// TIA Portal project "BasementLightControl" (V16)
// This program is an implementation of basement light system with 2 switch and 1 light.

(* hardware
DEVICE "S7-1200 station_1"  S7-1200 Station
   slot 0: "Rack_0"  S7-1200 Rack  Rack  V1.0
   slot 1: "PLC_1"  CPU 1211C DC/DC/DC  6ES7 211-1AE40-0XB0  V4.4
DEVICE "TP900 Comfort"  TP900 Comfort
   slot 0: "TP900 Comfort"  TP900 Comfort  6AV2 124-0JC01-0AX0  16.0.0.0
   slot 1: "HMI_RT_5"  TP900 Comfort  6AV2 124-0JC01-0AX0  16.0.0.0
   slot 5: "TP900 Comfort._CP_1"  PROFINET Interface  16.0.0.0
      slot 1: "PROFINET Interface_1"  PROFINET Interface
         slot 1: "Port_1"  Port
         slot 2: "Port_2"  Port
   slot 7: "TP900 Comfort.I/DP_CP_1"  MPI/DP Interface  16.0.0.0
*)

// ===== PLC "PLC_1"  CPU 1211C DC/DC/DC =====

DATA_BLOCK "HMI_Inteface"   // DB1
{ S7_Optimized_Access := 'TRUE' }
VERSION : 0.1
   VAR
      upperSwitch : Bool;   // toggle switch for upper level switch control
      lowerSwitch : Bool;   // toggle switch for lower level switch control
      lightOutput : Bool;   // 0 = Light is ON; 1 = Light is OFF
   END_VAR
BEGIN
END_DATA_BLOCK

DATA_BLOCK "lightControl_DB"   // DB2
{ S7_Optimized_Access := 'TRUE' }
VERSION : 0.1
// stored: InstanceOfName lightControl
"lightControl"
BEGIN
END_DATA_BLOCK

FUNCTION_BLOCK "lightControl"   // FB1, LAD
{ S7_Optimized_Access := 'TRUE' }
VERSION : 0.1
   VAR_INPUT
      UpperLevelSwitch : Bool;
      LowerLevelSwitch : Bool;
   END_VAR
   VAR_OUTPUT
      Light : Bool;
   END_VAR
BEGIN

REGION Network 1: Set Light output when one of the switch is in ON Position
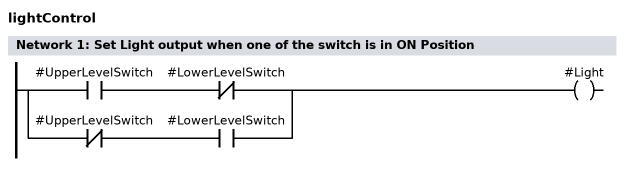
   RUNG wire#powerrail
      Contact( #UpperLevelSwitch )
      I_Contact( #LowerLevelSwitch )
      wire#w1
      Coil( #Light )
   END_RUNG
   RUNG wire#powerrail
      I_Contact( #UpperLevelSwitch )
      Contact( #LowerLevelSwitch )
   END_RUNG wire#w1
   // the same network as SCL:
   #Light := (#UpperLevelSwitch AND NOT #LowerLevelSwitch) OR (NOT #UpperLevelSwitch AND #LowerLevelSwitch);
END_REGION
END_FUNCTION_BLOCK

ORGANIZATION_BLOCK "Main"   // OB1, LAD, ProgramCycle
TITLE = "Main Program Sweep (Cycle)"
{ S7_Optimized_Access := 'TRUE' }
VERSION : 0.1
   VAR_INPUT
      Initial_Call : Bool;   // Initial call of this OB
      Remanence : Bool;   // =True, if remanent data are available
   END_VAR
BEGIN

REGION Network 1: Call Light Control FB
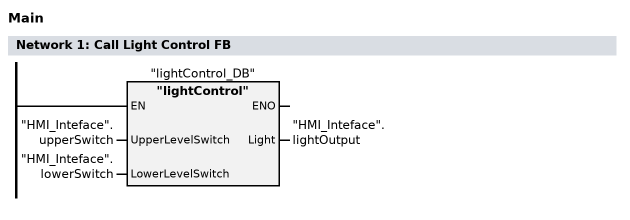
   RUNG wire#powerrail
      "lightControl_DB"(UpperLevelSwitch := "HMI_Inteface".upperSwitch, LowerLevelSwitch := "HMI_Inteface".lowerSwitch, Light => "HMI_Inteface".lightOutput)
   END_RUNG
   // the same network as SCL:
   "lightControl_DB"(UpperLevelSwitch := "HMI_Inteface".upperSwitch,   // "lightControl"
                     LowerLevelSwitch := "HMI_Inteface".lowerSwitch,
                     Light => "HMI_Inteface".lightOutput);
END_REGION
END_ORGANIZATION_BLOCK

(* ===== HMI "HMI_RT_5" =====
system functions are stored by id; their names below are inferred from use
connection "HMI_Connection_7": 
connection "HMI_Connection_1": ETHERNET, S7_1200_OMS

HMI tags "Template"
   "MainNavigationState" : Int, internal
   "SubNavigationState" : Int, internal
   "CurrentUserName" : WString[18], internal
   "DiagState" : Int, internal
   "PopUpBackground" : Bool, internal
   "UserName" : WString[20], internal
   "Password" : WString[20], internal
   "UserIsLoggedIn" : Bool, internal
   "CodeView" : Bool, internal
   "Brightness" : Int, internal
   "CurrentLanguage" : Bool, internal
   "CurrentRecipeName" : WString[30], internal
   "CurrentMachineState" : Int, internal
   "OptionPanelNavigationState" : Int, internal
   "ButtonDown" : Bool, internal
   "ThirdLevelNavigationState" : Int, internal
   "StartScreenName" : WString[60], internal
   "InScreenTabState" : Int, internal
   "DummyTagBool" : Bool, internal
   "DummyTagInt1" : Int, internal
   "DummyTagInt2" : Int, internal
   "DummyTagInt3" : Int, internal
   "DummyDeltaReal" : LReal, internal
   "DummTagReal1" : LReal, internal
   "DummyDeltaInt" : Int, internal

HMI tags "PLC_Tags"
   "HMI_Inteface_upperSwitch" : Bool = PLC HMI_Inteface.upperSwitch, 100 ms
   "HMI_Inteface_lowerSwitch" : Bool = PLC HMI_Inteface.lowerSwitch, 100 ms
   "HMI_Inteface_lightOutput" : Bool = PLC HMI_Inteface.lightOutput, 100 ms

text list "Machine State": 0 'Undefined / Kein Job'; 1 'Production / Produktion'; 2 'Startup / Anlauf'; 3 'Paused / Pausiert'; 4 'Stopped / Gestoppt'; 5 'Shutdown / Beenden'; 6 'Undefined / UNBEKANNT'

text list "timeRange": 1 'Hours / Stunden'; 2 'Days / Tage'; 3 'Weeks / Wochen'; 4 'Months / Monate'; 5 'Years / Jahre'

text list "MachineState_Farfield": 0..1 '???'; 1 'OK'; 2 'ERROR / FEHLER'; 3 'PAUSED / HALT'

text list "Foil Types": 0..1 '120 - 1mm - Transparent'; 1 '120 - 3mm - Transparent'; 2 '240 - 1mm - Transparent'; 3 '240 - 3mm - Transparent'

text list "FunctionState": 0 'Disabled / Deaktiviert'; 1 'Enabled / Aktiviert'

text list "GroundPos": 0 'No / Nein'; 1 'Yes / Ja'

text list "State": 0 'Off / Aus'; 1 'On / An'

graphic list "DiagState": 0 'DiagOkay'; 1 'DiagWarning_1'; 2 'DiagDefault'

graphic list "DiagState_1": 0 'DiagOkay_1'; 1 'DiagWarning'; 2 'DiagDefault'

graphic list "DiagState_2": 0 'DiagOkay_1'; 1 'DiagWarning'; 2 'DiagDefault'

graphic list "DiagState_3": 0 'DiagOkay_White'; 1 'DiagWarning_White'; 2 'Circle'

graphic list "State": 0..1 'OK'; 3 'Error'

graphic list "Machine": 1 'Grafik_Verpackung_Step1_Blink-off'; 2 'Grafik_Verpackung_Step2'; 3 'Grafik_Verpackung_Blink-on'; 6..7 'Grafik_Verpackung_Step1_Blink-off'

screen "20_Messages" 800x480, template "01_One_Nav_Level"
   on GenerateScreen: SetTag("MainNavigationState", 2)
   AlarmView "Alarm view_1" at 0,104 size 800x375
   GraphicView "Graphic view_2" at 0,0 size 800x480; Picture "PopUpBackground"
      Visibility <- "PopUpBackground"

screen "30_Diagnostics" 800x480, template "01_One_Nav_Level"
   on GenerateScreen: SetTag("MainNavigationState", 3)
   SysDiagControl "System diagnostics view_1" at 0,104 size 800x375
   GraphicView "Graphic view_2" at 0,0 size 800x480; Picture "PopUpBackground"
      Visibility <- "PopUpBackground"

screen "40_Settings" 800x480, template "02_Settings"
   on GenerateScreen: SetTag("MainNavigationState", 4)
   Slider "Template_Slider_1" at 320,133 size 300x30; Caption 'SIMATIC'
      on Change: function_e4c2bb66("Brightness")
      ProcessValue <- "Brightness"
   TextField "Template_Text field_1" at 180,136 size 92x24; Text 'Brightness / Helligkeit'
   GraphicView "Graphic view_2" at 0,0 size 800x480; Picture "PopUpBackground"
      Visibility <- "PopUpBackground"

screen "10_Startscreen" 800x480, template "01_One_Nav_Level"
   on GenerateScreen: "GetStartScreenName"(); "CheckCurrentUserName"(); SetTag("MainNavigationState", 1)
   GraphicView "Graphic view_2" at 0,0 size 800x480; Picture "PopUpBackground"
      Visibility <- "PopUpBackground"
   GraphicView "Graphic view_4" at 276,110 size 76x90; Picture "lighton"
      Visibility <- "HMI_Inteface_lightOutput"
   GraphicView "Graphic view_1" at 115,128 size 566x347; Picture "Stairs"
   Switch "Switch_1" at 10,108 size 64x169; CaptionText 'Upper'; TextOff 'OFF'; TextOn 'ON'
      ProcessValue <- "HMI_Inteface_upperSwitch"
   Switch "Switch_2" at 730,306 size 64x169; TextOn 'ON'; CaptionText 'Bottom'; TextOff 'OFF'
      ProcessValue <- "HMI_Inteface_lowerSwitch"
   GraphicView "Graphic view_3" at 276,110 size 76x90; Picture "lightoff"
      Visibility <- "HMI_Inteface_lightOutput"
   GraphicView "Graphic view_5" at 409,110 size 76x90; Picture "lighton"
      Visibility <- "HMI_Inteface_lightOutput"
   GraphicView "Graphic view_6" at 542,110 size 76x90; Picture "lighton"
      Visibility <- "HMI_Inteface_lightOutput"
   GraphicView "Graphic view_7" at 409,110 size 76x90; Picture "lightoff"
      Visibility <- "HMI_Inteface_lightOutput"
   GraphicView "Graphic view_8" at 542,110 size 76x90; Picture "lightoff"
      Visibility <- "HMI_Inteface_lightOutput"

Template "02_Two_Nav_Levels" 800x480
   GraphicView "gfxPrevScreenIcon" at 760,444 size 24x24; Picture "PrevScreen_Icon"
   Button "btnSubNav1" at 0,432 size 120x48; TextOff 'Overview / Übersicht'
      on Click: SetTag("SubNavigationState", 1)
   Button "btnSubNav2" at 120,432 size 120x48; TextOff 'Module 1 / Modul 1'
      on Click: SetTag("SubNavigationState", 2)
   Button "btnSubNav3" at 240,432 size 120x48; TextOff 'Module 2 / Modul 2'
      on Click: SetTag("SubNavigationState", 3)
   Button "btnSubNav4" at 360,432 size 120x48; TextOff 'Module 3 / Modul 3'
      on Click: SetTag("SubNavigationState", 4)
   Button "btnSubNav5" at 480,432 size 120x48; TextOff 'Module 4 / Modul 4'
      on Click: SetTag("SubNavigationState", 5)
   Button "btnSubNav6" at 600,432 size 120x48; TextOff 'Module 5 / Modul 5'
      on Click: SetTag("SubNavigationState", 6)
   Button "btnPreviousScreen" at 744,432 size 56x48; TextOff 'Text'
      on Click: function_efd93a16()
   Gauge "gaugeDiagStateUpdate" at 566,2 size 50x50; CaptionText 'SIMATIC'
      on Change: "CheckDiagState"()
      ProcessValue <- "@DiagnosticsIndicatorTag"
   TextField "txtTitleBar" at 16,8 size 495x32; Text 'Basement Light Control / Applikation'
   GraphicView "gfxNavigationIcon" at 761,15 size 23x19; Picture "Hamburger_Icon"
   Button "btnNavigation" at 744,0 size 56x48; TextOff 'Text'
      on Click: function_cf6f4242("GraphX_Slidein_Right", 1)
   TextField "txtStateHeadline" at 75,55 size 123x23; Text 'State / Status'
   TextField "txtRecipeHeadline" at 281,55 size 154x23; Text 'Current Recipe / Rezeptur'
   TextField "txtOperatorHeadline" at 527,55 size 129x23; Text 'Operator / Bediener'
   SymbolicIOField "ioState" at 75,72 size 119x30; TextOn '1'; TextOff '0'; TextList "Machine State"
      ProcessValue <- "CurrentMachineState"
   IOField "ioRecipe" at 281,72 size 158x30; FormatPattern ??????????????????????????????
      ProcessValue <- "CurrentRecipeName"
   IOField "ioOperator" at 527,72 size 126x30; FormatPattern ??????????????????
      ProcessValue <- "CurrentUserName"
   Button "btnState" at 202,56 size 40x40; TextOff '...'; PictureOff "More_Icon"
      on Click: "ShowOperatingModePopUp"()
   Button "btnRecipe" at 449,56 size 40x40; TextOff '...'; PictureOff "More_Icon"
      on Click: "ShowRecipePopUp"()
   Rectangle "rectState" at 0,48 size 56x56
      Appearance <- "CurrentMachineState"
   Rectangle "rectSystemDiagnosticsIndicator" at 744,48 size 56x56
      Appearance <- "DiagState"
   GraphicIOField "gioDiagState" at 756,60 size 32x32; PictureList "DiagState_3"
      ProcessValue <- "DiagState"
   Button "btnDiagState" at 744,48 size 56x56; TextOff 'Text'
      on Click: ActivateScreen("30_Diagnostics", 0)
   Button "btnOperator" at 669,56 size 40x40; TextOff '...'; PictureOff "More_Icon"
      on Click: "ShowLoginPopUp"()
   Button "btnStartscreen" at 0,0 size 250x45; TextOff 'Text'
      on Click: "ActivateStartScreen"()
   Button "btnSubNavActive1" at 0,432 size 120x48; TextOff 'Overview / Übersicht'
      Visibility <- "SubNavigationState"
   Button "btnSubNavActive2" at 120,432 size 120x48; TextOff 'Module 1 / Modul 1'
      Visibility <- "SubNavigationState"
   Button "btnSubNavActive3" at 240,432 size 120x48; TextOff 'Module 2 / Modul 2'
      Visibility <- "SubNavigationState"
   Button "btnSubNavActive4" at 360,432 size 120x48; TextOff 'Module 3 / Modul 3'
      Visibility <- "SubNavigationState"
   Button "btnSubNavActive5" at 480,432 size 120x48; TextOff 'Module 4 / Modul 4'
      Visibility <- "SubNavigationState"
   Button "btnSubNavActive6" at 600,432 size 120x48; TextOff 'Module 5 / Modul 5'
      Visibility <- "SubNavigationState"
   Rectangle "rectIndicatorActive1" at 0,475 size 120x5
      Visibility <- "SubNavigationState"
   Rectangle "rectIndicatorActive2" at 120,475 size 120x5
      Visibility <- "SubNavigationState"
   Rectangle "rectIndicatorActive3" at 240,475 size 120x5
      Visibility <- "SubNavigationState"
   Rectangle "rectIndicatorActive4" at 360,475 size 120x5
      Visibility <- "SubNavigationState"
   Rectangle "rectIndicatorActive5" at 480,475 size 120x5
      Visibility <- "SubNavigationState"
   Rectangle "rectIndicatorActive6" at 600,475 size 120x5
      Visibility <- "SubNavigationState"

Template "03_Three_Nav_Levels" 800x480
   Button "btnStartscreen" at 0,0 size 326x45; TextOff 'Text'
      on Click: "ActivateStartScreen"()
   Gauge "gaugeDiagStateUpdate" at 566,2 size 50x50; CaptionText 'SIMATIC'
      on Change: "CheckDiagState"()
      ProcessValue <- "@DiagnosticsIndicatorTag"
   TextField "txtTitleBar" at 16,8 size 495x32; Text 'Basement Light Control / Applikation'
   GraphicView "gfxNavigationIcon" at 761,15 size 23x19; Picture "Hamburger_Icon"
   Button "btnNavigation" at 744,0 size 56x48; TextOff 'Text'
      on Click: function_cf6f4242("GraphX_Slidein_Right", 1)
   Rectangle "rectSystemDiagnosticsIndicator" at 744,48 size 56x56
      Appearance <- "DiagState"
   GraphicIOField "gioDiagState" at 756,60 size 32x32; PictureList "DiagState_3"
      ProcessValue <- "DiagState"
   Button "btnDiagState" at 744,48 size 56x56; TextOff 'Text'
      on Click: ActivateScreen("30_Diagnostics", 0)
   TextField "txtStateHeadline" at 75,55 size 123x23; Text 'State / Status'
   TextField "txtOperatorHeadline" at 527,55 size 129x23; Text 'Operator / Bediener'
   SymbolicIOField "ioState" at 75,72 size 119x30; TextOn '1'; TextOff '0'; TextList "Machine State"
      ProcessValue <- "CurrentMachineState"
   IOField "ioOperator" at 527,72 size 126x30; FormatPattern ??????????????????
      ProcessValue <- "CurrentUserName"
   Button "btnState" at 202,56 size 40x40; TextOff '...'; PictureOff "More_Icon"
      on Click: "ShowOperatingModePopUp"()
   Button "btnOperator" at 669,56 size 40x40; TextOff '...'; PictureOff "More_Icon"
      on Click: "ShowLoginPopUp"()
   Rectangle "rectState" at 0,48 size 56x56
      Appearance <- "CurrentMachineState"
   TextField "txtRecipeHeadline" at 281,55 size 154x23; Text 'Current Recipe / Rezeptur'
   IOField "ioRecipe" at 281,72 size 158x30; FormatPattern ??????????????????????????????
      ProcessValue <- "CurrentRecipeName"
   Button "btnRecipe" at 449,56 size 40x40; TextOff '...'; PictureOff "More_Icon"
      on Click: "ShowRecipePopUp"()
   Button "btnThirdLevel4btnOff1" at 0,104 size 56x83; TextOff 'Text'
   Button "btnThirdLevel4btnOff2" at 0,186 size 56x83; TextOff 'Text'
   Button "btnThirdLevel4btnOff3" at 0,268 size 56x83; TextOff 'Text'
   Button "btnThirdLevel4btnOff4" at 0,350 size 56x82; TextOff 'Text'
   Button "btnThirdLevel4btnOn1" at 0,187 size 56x81; TextOff 'Text'
      Visibility <- "ThirdLevelNavigationState"
   Button "btnThirdLevel4btnOn2" at 0,104 size 56x82; TextOff 'Text'
      Visibility <- "ThirdLevelNavigationState"
   Button "btnThirdLevel4btnOn3" at 0,269 size 56x81; TextOff 'Text'
      Visibility <- "ThirdLevelNavigationState"
   Button "btnThirdLevel4btnOn4" at 0,351 size 56x81; TextOff 'Text'
      Visibility <- "ThirdLevelNavigationState"
   Rectangle "rectIndicator4btnActive1" at 0,104 size 5x82
      Visibility <- "ThirdLevelNavigationState"
   Rectangle "rectIndicator4btnActive2" at 0,187 size 5x81
      Visibility <- "ThirdLevelNavigationState"
   Rectangle "rectIndicator4btnActive3" at 0,269 size 5x81
      Visibility <- "ThirdLevelNavigationState"
   Rectangle "rectIndicator4btnActive4" at 0,351 size 5x81
      Visibility <- "ThirdLevelNavigationState"
   Button "btnSubNav1" at 0,432 size 120x48; TextOff 'Overview / Übersicht'
      on Click: SetTag("SubNavigationState", 1)
   Button "btnSubNav2" at 120,432 size 120x48; TextOff 'Module 1 / Modul 1'
      on Click: SetTag("SubNavigationState", 2)
   Button "btnSubNav3" at 240,432 size 120x48; TextOff 'Module 2 / Modul 2'
      on Click: SetTag("SubNavigationState", 3)
   Button "btnSubNav4" at 360,432 size 120x48; TextOff 'Module 3 / Modul 3'
      on Click: SetTag("SubNavigationState", 4)
   Button "btnSubNav5" at 480,432 size 120x48; TextOff 'Module 4 / Modul 4'
      on Click: SetTag("SubNavigationState", 5)
   Button "btnSubNav6" at 600,432 size 120x48; TextOff 'Module 5 / Modul 5'
      on Click: SetTag("SubNavigationState", 6)
   GraphicView "gfxPrevScreenIcon" at 760,444 size 24x24; Picture "PrevScreen_Icon"
   Button "btnPreviousScreen" at 744,432 size 56x48; TextOff 'Text'
      on Click: function_efd93a16()
   Button "btnSubNavActive1" at 0,432 size 120x48; TextOff 'Overview / Übersicht'
      Visibility <- "SubNavigationState"
   Button "btnSubNavActive2" at 120,432 size 120x48; TextOff 'Module 1 / Modul 1'
      Visibility <- "SubNavigationState"
   Button "btnSubNavActive3" at 240,432 size 120x48; TextOff 'Module 2 / Modul 2'
      Visibility <- "SubNavigationState"
   Button "btnSubNavActive4" at 360,432 size 120x48; TextOff 'Module 3 / Modul 3'
      Visibility <- "SubNavigationState"
   Button "btnSubNavActive5" at 480,432 size 120x48; TextOff 'Module 4 / Modul 4'
      Visibility <- "SubNavigationState"
   Button "btnSubNavActive6" at 600,432 size 120x48; TextOff 'Module 5 / Modul 5'
      Visibility <- "SubNavigationState"
   Rectangle "rectIndicatorActive1" at 0,475 size 120x5
      Visibility <- "SubNavigationState"
   Rectangle "rectIndicatorActive2" at 120,475 size 120x5
      Visibility <- "SubNavigationState"
   Rectangle "rectIndicatorActive3" at 240,475 size 120x5
      Visibility <- "SubNavigationState"
   Rectangle "rectIndicatorActive4" at 360,475 size 120x5
      Visibility <- "SubNavigationState"
   Rectangle "rectIndicatorActive5" at 480,475 size 120x5
      Visibility <- "SubNavigationState"
   Rectangle "rectIndicatorActive6" at 600,475 size 120x5
      Visibility <- "SubNavigationState"

Template "03_Three_Nav_Levels_w_OptionPanel" 800x480
   Button "btnStartscreen" at 0,0 size 326x45; TextOff 'Text'
      on Click: "ActivateStartScreen"()
   Gauge "gaugeDiagStateUpdate" at 566,2 size 50x50; CaptionText 'SIMATIC'
      on Change: "CheckDiagState"()
      ProcessValue <- "@DiagnosticsIndicatorTag"
   TextField "txtTitleBar" at 16,8 size 495x32; Text 'Basement Light Control / Applikation'
   GraphicView "gfxNavigationIcon" at 761,15 size 23x19; Picture "Hamburger_Icon"
   Button "btnNavigation" at 744,0 size 56x48; TextOff 'Text'
      on Click: function_cf6f4242("GraphX_Slidein_Right", 1)
   Rectangle "rectSystemDiagnosticsIndicator" at 744,48 size 56x56
      Appearance <- "DiagState"
   GraphicIOField "gioDiagState" at 756,60 size 32x32; PictureList "DiagState_3"
      ProcessValue <- "DiagState"
   Button "btnDiagState" at 744,48 size 56x56; TextOff 'Text'
      on Click: ActivateScreen("30_Diagnostics", 0)
   TextField "txtStateHeadline" at 75,55 size 123x23; Text 'State / Status'
   TextField "txtOperatorHeadline" at 527,55 size 129x23; Text 'Operator / Bediener'
   SymbolicIOField "ioState" at 75,72 size 119x30; TextOn '1'; TextOff '0'; TextList "Machine State"
      ProcessValue <- "CurrentMachineState"
   IOField "ioOperator" at 527,72 size 126x30; FormatPattern ??????????????????
      ProcessValue <- "CurrentUserName"
   Button "btnState" at 202,56 size 40x40; TextOff '...'; PictureOff "More_Icon"
      on Click: "ShowOperatingModePopUp"()
   Button "btnOperator" at 669,56 size 40x40; TextOff '...'; PictureOff "More_Icon"
      on Click: "ShowLoginPopUp"()
   Rectangle "rectState" at 0,48 size 56x56
      Appearance <- "CurrentMachineState"
   TextField "txtRecipeHeadline" at 281,55 size 154x23; Text 'Current Recipe / Rezeptur'
   IOField "ioRecipe" at 281,72 size 158x30; FormatPattern ??????????????????????????????
      ProcessValue <- "CurrentRecipeName"
   Button "btnRecipe" at 449,56 size 40x40; TextOff '...'; PictureOff "More_Icon"
      on Click: "ShowRecipePopUp"()
   Button "btnThirdLevelOff1" at 0,104 size 56x83; TextOff 'Text'
   Button "btnThirdLevelOff2" at 0,186 size 56x83; TextOff 'Text'
   Button "btnThirdLevelOff3" at 0,268 size 56x83; TextOff 'Text'
   Button "btnThirdLevelOff4" at 0,350 size 56x82; TextOff 'Text'
   Button "btnThirdLevelOn1" at 0,187 size 56x81; TextOff 'Text'
      Visibility <- "ThirdLevelNavigationState"
   Button "btnThirdLevelOn2" at 0,104 size 56x82; TextOff 'Text'
      Visibility <- "ThirdLevelNavigationState"
   Button "btnThirdLevelOn3" at 0,269 size 56x81; TextOff 'Text'
      Visibility <- "ThirdLevelNavigationState"
   Button "btnThirdLevelOn4" at 0,351 size 56x81; TextOff 'Text'
      Visibility <- "ThirdLevelNavigationState"
   Rectangle "rectIndicatorActive1_1" at 0,104 size 5x82
      Visibility <- "ThirdLevelNavigationState"
   Rectangle "rectIndicatorActive1_2" at 0,187 size 5x81
      Visibility <- "ThirdLevelNavigationState"
   Rectangle "rectIndicatorActive1_3" at 0,269 size 5x81
      Visibility <- "ThirdLevelNavigationState"
   Rectangle "rectIndicatorActive1_4" at 0,351 size 5x81
      Visibility <- "ThirdLevelNavigationState"
   Button "btnOption1btn1" at 744,104 size 56x328; TextOff 'Text'; PictureOff "ManFunctions_Off"; PictureOn "ManFunctions_Off"
      on Click: "ShowOptionPanelPopUp"()
   Button "btnSubNav1" at 0,432 size 120x48; TextOff 'Overview / Übersicht'
      on Click: SetTag("SubNavigationState", 1)
   Button "btnSubNav2" at 120,432 size 120x48; TextOff 'Module 1 / Modul 1'
      on Click: SetTag("SubNavigationState", 2)
   Button "btnSubNav3" at 240,432 size 120x48; TextOff 'Module 2 / Modul 2'
      on Click: SetTag("SubNavigationState", 3)
   Button "btnSubNav4" at 360,432 size 120x48; TextOff 'Module 3 / Modul 3'
      on Click: SetTag("SubNavigationState", 4)
   Button "btnSubNav5" at 480,432 size 120x48; TextOff 'Module 4 / Modul 4'
      on Click: SetTag("SubNavigationState", 5)
   Button "btnSubNav6" at 600,432 size 120x48; TextOff 'Module 5 / Modul 5'
      on Click: SetTag("SubNavigationState", 6)
   GraphicView "gfxPrevScreenIcon" at 760,444 size 24x24; Picture "PrevScreen_Icon"
   Button "btnPreviousScreen" at 744,432 size 56x48; TextOff 'Text'
      on Click: function_efd93a16()
   Button "btnSubNavActive1" at 0,432 size 120x48; TextOff 'Overview / Übersicht'
      Visibility <- "SubNavigationState"
   Button "btnSubNavActive2" at 120,432 size 120x48; TextOff 'Module 1 / Modul 1'
      Visibility <- "SubNavigationState"
   Button "btnSubNavActive3" at 240,432 size 120x48; TextOff 'Module 2 / Modul 2'
      Visibility <- "SubNavigationState"
   Button "btnSubNavActive4" at 360,432 size 120x48; TextOff 'Module 3 / Modul 3'
      Visibility <- "SubNavigationState"
   Button "btnSubNavActive5" at 480,432 size 120x48; TextOff 'Module 4 / Modul 4'
      Visibility <- "SubNavigationState"
   Button "btnSubNavActive6" at 600,432 size 120x48; TextOff 'Module 5 / Modul 5'
      Visibility <- "SubNavigationState"
   Rectangle "rectIndicatorActive1" at 0,475 size 120x5
      Visibility <- "SubNavigationState"
   Rectangle "rectIndicatorActive2" at 120,475 size 120x5
      Visibility <- "SubNavigationState"
   Rectangle "rectIndicatorActive3" at 240,475 size 120x5
      Visibility <- "SubNavigationState"
   Rectangle "rectIndicatorActive4" at 360,475 size 120x5
      Visibility <- "SubNavigationState"
   Rectangle "rectIndicatorActive5" at 480,475 size 120x5
      Visibility <- "SubNavigationState"
   Rectangle "rectIndicatorActive6" at 600,475 size 120x5
      Visibility <- "SubNavigationState"

Template "01_One_Nav_Level" 800x480
   Rectangle "rectSystemDiagnosticsIndicator" at 744,48 size 56x56
      Appearance <- "DiagState"
   GraphicIOField "gioDiagState" at 756,60 size 32x32; PictureList "DiagState_3"
      ProcessValue <- "DiagState"
   Button "btnDiagState" at 744,48 size 56x56; TextOff 'Text'
      on Click: ActivateScreen("30_Diagnostics", 0)
   TextField "txtStateHeadline" at 75,55 size 123x23; Text 'State / Status'
   TextField "txtOperatorHeadline" at 527,55 size 129x23; Text 'Operator / Bediener'
   SymbolicIOField "ioState" at 75,72 size 119x30; TextOn '1'; TextOff '0'; TextList "Machine State"
      ProcessValue <- "CurrentMachineState"
   IOField "ioOperator" at 527,72 size 126x30; FormatPattern ??????????????????
      ProcessValue <- "CurrentUserName"
   Button "btnState" at 202,56 size 40x40; TextOff '...'; PictureOff "More_Icon"
      on Click: "ShowOperatingModePopUp"()
   Button "btnOperator" at 669,56 size 40x40; TextOff '...'; PictureOff "More_Icon"
      on Click: "ShowLoginPopUp"()
   Rectangle "rectState" at 0,48 size 56x56
      Appearance <- "CurrentMachineState"
   TextField "txtRecipeHeadline" at 281,55 size 154x23; Text 'Current Recipe / Rezeptur'
   IOField "ioRecipe" at 281,72 size 158x30; FormatPattern ??????????????????????????????
      ProcessValue <- "CurrentRecipeName"
   Button "btnRecipe" at 449,56 size 40x40; TextOff '...'; PictureOff "More_Icon"
      on Click: "ShowRecipePopUp"()
   Gauge "gaugeDiagStateUpdate" at 566,2 size 50x50; CaptionText 'SIMATIC'
      on Change: "CheckDiagState"()
      ProcessValue <- "@DiagnosticsIndicatorTag"
   GraphicView "gfxNavigationIcon" at 761,15 size 23x19; Picture "Hamburger_Icon"
   Button "btnNavigation" at 744,0 size 56x48; TextOff 'Text'
      on Click: function_cf6f4242("GraphX_Slidein_Right", 1)
   TextField "txtTitleBar" at 16,8 size 495x32; Text 'Basement Light Control / Applikation'
   Button "btnStartscreen" at 0,0 size 250x45; TextOff 'Text'
      on Click: "ActivateStartScreen"()

Template "02_Two_Nav_Levels_Large_Text" 800x480
   Gauge "gaugeDiagStateUpdate" at 566,2 size 50x50; CaptionText 'SIMATIC'
      on Change: "CheckDiagState"()
      ProcessValue <- "@DiagnosticsIndicatorTag"
   TextField "txtTitleBar" at 16,8 size 495x32; Text 'Basement Light Control / Applikation'
   GraphicView "gfxNavigationIcon" at 761,15 size 23x19; Picture "Hamburger_Icon"
   Button "btnNavigation" at 744,0 size 56x48; TextOff 'Text'
      on Click: function_cf6f4242("GraphX_Slidein_Right", 1)
   TextField "txtStateHeadline" at 75,55 size 123x23; Text 'State / Status'
   TextField "txtRecipeHeadline" at 281,55 size 154x23; Text 'Current Recipe / Rezeptur'
   TextField "txtOperatorHeadline" at 527,55 size 129x23; Text 'Operator / Bediener'
   SymbolicIOField "ioState" at 75,72 size 119x30; TextOn '1'; TextOff '0'; TextList "Machine State"
      ProcessValue <- "CurrentMachineState"
   IOField "ioRecipe" at 281,72 size 158x30; FormatPattern ??????????????????????????????
      ProcessValue <- "CurrentRecipeName"
   IOField "ioOperator" at 527,72 size 126x30; FormatPattern ??????????????????
      ProcessValue <- "CurrentUserName"
   Button "btnState" at 202,56 size 40x40; TextOff '...'; PictureOff "More_Icon"
      on Click: "ShowOperatingModePopUp"()
   Button "btnRecipe" at 449,56 size 40x40; TextOff '...'; PictureOff "More_Icon"
      on Click: "ShowRecipePopUp"()
   Rectangle "rectState" at 0,48 size 56x56
      Appearance <- "CurrentMachineState"
   GraphicView "gfxPrevScreenIcon" at 760,444 size 24x24; Picture "PrevScreen_Icon"
   Button "btnPreviousScreen" at 744,432 size 56x48; TextOff 'Text'
      on Click: function_efd93a16()
   TextField "txtCurrentStateInfo" at 16,444 size 505x24; Text 'Optional Text about current state / Optional. Text aktueller Status'
   Rectangle "rectSystemDiagnosticsIndicator" at 744,48 size 56x56
      Appearance <- "DiagState"
   GraphicIOField "gioDiagState" at 756,60 size 32x32; PictureList "DiagState_3"
      ProcessValue <- "DiagState"
   Button "btnDiagState" at 744,48 size 56x56; TextOff 'Text'
      on Click: ActivateScreen("30_Diagnostics", 0)
   Button "btnOperator" at 669,56 size 40x40; TextOff '...'; PictureOff "More_Icon"
      on Click: "ShowLoginPopUp"()
   Button "btnStartscreen" at 0,0 size 250x45; TextOff 'Text'
      on Click: "ActivateStartScreen"()
   Rectangle "rectSubNavigation1" at 0,104 size 264x83
      Appearance <- "ThirdLevelNavigationState"
   Rectangle "rectSubNavigation2" at 0,186 size 264x83
      Appearance <- "ThirdLevelNavigationState"
   Rectangle "rectSubNavigation3" at 0,268 size 264x83
      Appearance <- "ThirdLevelNavigationState"
   Rectangle "rectSubNavigation4" at 0,350 size 264x82
      Appearance <- "ThirdLevelNavigationState"
   TextField "txtOption1" at 16,120 size 232x24; Text 'Option 1'
   IOField "ioValueOption1" at 16,152 size 236x24; FormatPattern ??????????????????????????????????????????????????
   TextField "txtOption2" at 16,202 size 232x24; Text 'Option 2'
   IOField "ioValueOption2" at 16,234 size 236x24; FormatPattern ??????????????????????????????????????????????????
   TextField "txtOption3" at 16,284 size 232x24; Text 'Option 3'
   IOField "ioValueOption3" at 16,316 size 236x24; FormatPattern ??????????????????????????????????????????????????
   TextField "txtOption4" at 16,366 size 232x24; Text 'Option 4'
   IOField "ioValueOption4" at 16,398 size 236x24; FormatPattern ??????????????????????????????????????????????????
   Button "btnSubNavigation1" at 0,104 size 264x83; TextOff 'Text'
      on Click: SetTag("ThirdLevelNavigationState", 1)
   Button "btnSubNavigation2" at 0,186 size 264x83; TextOff 'Text'
      on Click: SetTag("ThirdLevelNavigationState", 2)
   Button "btnSubNavigation3" at 0,268 size 264x83; TextOff 'Text'
      on Click: SetTag("ThirdLevelNavigationState", 3)
   Button "btnSubNavigation4" at 0,350 size 264x83; TextOff 'Text'
      on Click: SetTag("ThirdLevelNavigationState", 4)

Template "02_Two_Nav_Levels_Text" 800x480
   Button "btnSubNav1" at 0,120 size 136x56; TextOn 'Item 1'; TextOff 'Item 1'
      on Click: SetTag("SubNavigationState", 1)
   Button "btnSubNav2" at 0,175 size 136x56; TextOn 'Item 2'; TextOff 'Item 2'
      on Click: SetTag("SubNavigationState", 2)
   Button "btnSubNav3" at 0,230 size 136x60; TextOn 'Item 3'; TextOff 'Item 3'
      on Click: SetTag("SubNavigationState", 3)
   GraphicView "gfxRuntimeStop" at 57,443 size 23x28; Picture "Power_dark"
   Button "btnRuntimeStop" at 0,432 size 136x48; TextOff 'Text'
      on Click: StopRuntime(0)
   Button "btnSubNav3_1" at 0,289 size 136x60; TextOn 'Item 4'; TextOff 'Item 4'
      on Click: SetTag("SubNavigationState", 4)
   Button "btnSubNav3_2" at 0,348 size 136x60; TextOn 'Item 5'; TextOff 'Item 5'
      on Click: SetTag("SubNavigationState", 5)
   Button "btnSubNavActive3" at 0,230 size 136x60; TextOff 'Item 3'
      Visibility <- "SubNavigationState"
   Button "btnSubNavActive1" at 0,120 size 136x56; TextOff 'Item 1'
      Visibility <- "SubNavigationState"
   Button "btnSubNavActive2" at 0,175 size 136x56; TextOff 'Item 2'
      Visibility <- "SubNavigationState"
   Rectangle "rectIndicatorActive3" at 0,230 size 5x60
      Visibility <- "SubNavigationState"
   Rectangle "rectIndicatorActive1" at 0,120 size 5x56
      Visibility <- "SubNavigationState"
   Rectangle "rectIndicatorActive2" at 0,175 size 5x56
      Visibility <- "SubNavigationState"
   Button "btnSubNavActive3_1" at 0,290 size 136x60; TextOff 'Item 4'
      Visibility <- "SubNavigationState"
   Rectangle "rectIndicatorActive3_1" at 0,290 size 5x60
      Visibility <- "SubNavigationState"
   Button "btnSubNavActive3_2" at 0,350 size 136x60; TextOff 'Item 5'
      Visibility <- "SubNavigationState"
   Rectangle "rectIndicatorActive3_2" at 0,350 size 5x60
      Visibility <- "SubNavigationState"
   Gauge "gaugeDiagStateUpdate" at 566,2 size 50x50; CaptionText 'SIMATIC'
      on Change: "CheckDiagState"()
      ProcessValue <- "@DiagnosticsIndicatorTag"
   GraphicView "gfxNavigationIcon" at 761,15 size 23x19; Picture "Hamburger_Icon"
   Button "btnNavigation" at 744,0 size 56x48; TextOff 'Text'
      on Click: function_cf6f4242("GraphX_Slidein_Right", 1)
   TextField "txtTitleBar" at 16,8 size 495x32; Text 'Basement Light Control / Applikation'
   Button "btnStartscreen" at 0,0 size 250x45; TextOff 'Text'
      on Click: "ActivateStartScreen"()
   TextField "txtStateHeadline" at 75,55 size 123x23; Text 'State / Status'
   TextField "txtOperatorHeadline" at 527,55 size 129x23; Text 'Operator / Bediener'
   SymbolicIOField "ioState" at 75,72 size 119x30; TextOn '1'; TextOff '0'; TextList "Machine State"
      ProcessValue <- "CurrentMachineState"
   IOField "ioOperator" at 527,72 size 126x30; FormatPattern ??????????????????
      ProcessValue <- "CurrentUserName"
   Button "btnState" at 202,56 size 40x40; TextOff '...'; PictureOff "More_Icon"
      on Click: "ShowOperatingModePopUp"()
   Button "btnOperator" at 669,56 size 40x40; TextOff '...'; PictureOff "More_Icon"
      on Click: "ShowLoginPopUp"()
   Rectangle "rectState" at 0,48 size 56x56
      Appearance <- "CurrentMachineState"
   TextField "txtRecipeHeadline" at 281,55 size 154x23; Text 'Current Recipe / Rezeptur'
   IOField "ioRecipe" at 281,72 size 158x30; FormatPattern ??????????????????????????????
      ProcessValue <- "CurrentRecipeName"
   Button "btnRecipe" at 449,56 size 40x40; TextOff '...'; PictureOff "More_Icon"
      on Click: "ShowRecipePopUp"()
   Rectangle "rectSystemDiagnosticsIndicator" at 744,48 size 56x56
      Appearance <- "DiagState"
   GraphicIOField "gioDiagState" at 756,60 size 32x32; PictureList "DiagState_3"
      ProcessValue <- "DiagState"
   Button "btnDiagState" at 744,48 size 56x56; TextOff 'Text'
      on Click: ActivateScreen("30_Diagnostics", 0)

Template "02_Settings" 800x480
   Button "btnSubNav1" at 0,120 size 136x56; TextOn 'Display'; TextOff 'Display'
      on Click: SetTag("SubNavigationState", 1)
   GraphicView "gfxRuntimeStop" at 57,443 size 23x28; Picture "Power_dark"
   Button "btnRuntimeStop" at 0,432 size 136x48; TextOff 'Text'
      on Click: StopRuntime(0)
   Button "btnSubNavActive1" at 0,120 size 136x56; TextOn 'Display'; TextOff 'Display'
      Visibility <- "SubNavigationState"
   Rectangle "rectIndicatorActive1" at 0,120 size 5x56
      Visibility <- "SubNavigationState"
   Gauge "gaugeDiagStateUpdate" at 566,2 size 50x50; CaptionText 'SIMATIC'
      on Change: "CheckDiagState"()
      ProcessValue <- "@DiagnosticsIndicatorTag"
   GraphicView "gfxNavigationIcon" at 761,15 size 23x19; Picture "Hamburger_Icon"
   Button "btnNavigation" at 744,0 size 56x48; TextOff 'Text'
      on Click: function_cf6f4242("GraphX_Slidein_Right", 1)
   TextField "txtTitleBar" at 16,8 size 495x32; Text 'Basement Light Control / Applikation'
   Button "btnStartscreen" at 0,0 size 250x45; TextOff 'Text'
      on Click: "ActivateStartScreen"()
   TextField "txtStateHeadline" at 75,55 size 123x23; Text 'State / Status'
   TextField "txtOperatorHeadline" at 527,55 size 129x23; Text 'Operator / Bediener'
   SymbolicIOField "ioState" at 75,72 size 119x30; TextOn '1'; TextOff '0'; TextList "Machine State"
      ProcessValue <- "CurrentMachineState"
   IOField "ioOperator" at 527,72 size 126x30; FormatPattern ??????????????????
      ProcessValue <- "CurrentUserName"
   Button "btnState" at 202,56 size 40x40; TextOff '...'; PictureOff "More_Icon"
      on Click: "ShowOperatingModePopUp"()
   Button "btnOperator" at 669,56 size 40x40; TextOff '...'; PictureOff "More_Icon"
      on Click: "ShowLoginPopUp"()
   Rectangle "rectState" at 0,48 size 56x56
      Appearance <- "CurrentMachineState"
   TextField "txtRecipeHeadline" at 281,55 size 154x23; Text 'Current Recipe / Rezeptur'
   IOField "ioRecipe" at 281,72 size 158x30; FormatPattern ??????????????????????????????
      ProcessValue <- "CurrentRecipeName"
   Button "btnRecipe" at 449,56 size 40x40; TextOff '...'; PictureOff "More_Icon"
      on Click: "ShowRecipePopUp"()
   Rectangle "rectSystemDiagnosticsIndicator" at 744,48 size 56x56
      Appearance <- "DiagState"
   GraphicIOField "gioDiagState" at 756,60 size 32x32; PictureList "DiagState_3"
      ProcessValue <- "DiagState"
   Button "btnDiagState" at 744,48 size 56x56; TextOff 'Text'
      on Click: ActivateScreen("30_Diagnostics", 0)

PopupScreen "Template_Logon" 320x352
   on ClearScreen: ResetBit("PopUpBackground")
   on GenerateScreen: SetBit("PopUpBackground")
   TextField "Template_Text field_1" at 16,0 size 215x40; Text 'Login'
   Button "Button_2" at 16,240 size 288x40; TextOn 'LOGIN / ANMELDEN'; TextOff 'LOGIN / ANMELDEN'
      on Click: function_a9b89908("Password", "UserName"); function_efd93a16("Template_Logon", 0, 0, 0, -1, 1)
   IOField "I/O field_1" at 16,84 size 288x40; FormatPattern ??????????????????????????????
      ProcessValue <- "UserName"
   TextField "Text field_1" at 16,56 size 288x24; Text 'User Name / Name'
   IOField "I/O field_2" at 16,168 size 288x40; FormatPattern ??????????????????????????????
      ProcessValue <- "Password"
   TextField "Text field_2" at 16,140 size 288x24; Text 'Password / Passwort'
   Button "Button_1" at 16,296 size 288x40; TextOn 'CLOSE / SCHLIESSEN'; TextOff 'CLOSE / SCHLIESSEN'
      on Click: function_efd93a16("Template_Logon", 0, 0, 0, -1, 1)
      on Press: function_b14e0dd5("ButtonDown", 0)
      Appearance <- "ButtonDown"

PopupScreen "Template_Logon_Logoff" 320x352
   on ClearScreen: ResetBit("PopUpBackground")
   on GenerateScreen: SetBit("PopUpBackground")
   TextField "Template_Text field_1" at 16,0 size 215x40; Text 'Login'
   Button "Button_2" at 16,240 size 136x40; TextOn 'LOG OFF / ABMELDEN'; TextOff 'LOG OFF / ABMELDEN'
      on Click: function_f23ef4c9()
   IOField "I/O field_1" at 16,84 size 288x40; FormatPattern ??????????????????????????????
      ProcessValue <- "UserName"
   TextField "Text field_1" at 16,56 size 288x24; Text 'User Name / Name'
   IOField "I/O field_2" at 16,168 size 288x40; FormatPattern ??????????????????????????????
      ProcessValue <- "Password"
   TextField "Text field_2" at 16,140 size 288x24; Text 'Password / Passwort'
   Button "Button_1" at 16,296 size 288x40; TextOn 'CLOSE / SCHLIESSEN'; TextOff 'CLOSE / SCHLIESSEN'
      on Click: function_efd93a16("Template_Logon_Logoff", 0, 0, 0, -1, 1)
      on Press: function_b14e0dd5("ButtonDown", 0)
      Appearance <- "ButtonDown"
   Button "Button_3" at 168,240 size 136x40; TextOn 'LOGIN / ANMELDEN'; TextOff 'LOGIN / ANMELDEN'
      on Click: function_a9b89908("Password", "UserName"); function_efd93a16("Template_Logon_Logoff", 0, 0, 0, -1, 1)

PopupScreen "Template_Operating_Mode" 424x360
   on ClearScreen: ResetBit("PopUpBackground")
   on GenerateScreen: SetBit("PopUpBackground")
   TextField "Template_Text field_1" at 14,0 size 336x40; Text 'Operating Mode / Betriebsmodus'
   Button "Button_1" at 80,304 size 260x40; TextOn 'CLOSE / SCHLIESSEN'; TextOff 'CLOSE / SCHLIESSEN'
      on Click: function_efd93a16("Template_Operating_Mode", 0, 0, 0, -1, 1)
      on Press: function_b14e0dd5("ButtonDown", 0)
      Appearance <- "ButtonDown"
   Button "Button_2" at 352,66 size 40x40; TextOff 'Text'; PictureOff "More_Icon"; PictureOn "More_Icon"
   Button "Button_3" at 352,130 size 40x40; TextOff 'Text'; PictureOff "More_Icon"; PictureOn "More_Icon"
   Button "Button_4" at 28,210 size 82x48; TextOff 'Start'
   Button "Button_5" at 123,210 size 82x48; TextOff 'Stop'
   Button "Button_6" at 218,210 size 82x48; TextOff 'Reset'
   Button "Button_7" at 314,210 size 82x48; TextOff 'Hold'
   TextField "txtParameter7_3" at 32,63 size 163x24; Text 'Current Mode'
   IOField "ioParameter17_3" at 32,81 size 301x40; FormatPattern ?????????????????????????
   TextField "txtParameter7_1" at 32,127 size 163x24; Text 'Current State'
   IOField "ioParameter17_1" at 32,145 size 301x40; FormatPattern ?????????????????????????

PopupScreen "Template_Recipe" 700x420
   on ClearScreen: ResetBit("PopUpBackground")
   on GenerateScreen: SetBit("PopUpBackground")
   TextField "Template_Text field_1" at 14,0 size 500x40; Text 'Recipe / Rezeptur'
   Button "Button_1" at 220,364 size 260x40; TextOn 'CLOSE / SCHLIESSEN'; TextOff 'CLOSE / SCHLIESSEN'
      on Click: function_efd93a16("Template_Recipe", 0, 0, 0, -1, 1)
      on Press: function_b14e0dd5("ButtonDown", 0)
      Appearance <- "ButtonDown"
   RecipeView "Rezepturanzeige_1" at 0,40 size 698x320

PopupScreen "OptionPanel_4_Buttons" 400x328
   GraphicView "gfxOptionPanel" at 80,30 size 18x12; Picture "ManFunctions_Off"
   TextField "textOptionPanelTitle" at 108,16 size 260x40; Text 'Option Panel Title / Titel Option Panel'
   Button "btnOptionPanelClose" at 0,0 size 40x328; TextOff 'Text'; PictureOff "Jog_Forward"
      on Press: function_efd93a16("OptionPanel_4_Buttons", 0, 0, 0, 2, 2)
   Button "btnOption1" at 80,72 size 240x40; TextOn 'Option 1'; TextOff 'Option 1 / Move to Home Position'
   Button "btnOption2" at 80,128 size 240x40; TextOn 'Option 2'; TextOff 'Option 2 / Move to Home Position'
   Button "btnOption3" at 80,184 size 240x40; TextOn 'Option 3'; TextOff 'Option 3 / RESET'
   Button "btnOption4" at 80,240 size 240x40; TextOn 'Option 4'; TextOff 'Option 4 / RESET'

SlideinScreen "GraphX_Slidein_Right" 220x480
   Button "Button_1" at 0,78 size 220x60; TextOn 'Menu Item 1'; TextOff 'Startscreen / Startseite'
      on Click: ActivateScreen("10_Startscreen", 0)
      Appearance <- "MainNavigationState"
   Button "Button_2" at 0,140 size 220x60; TextOn 'Menu Item 2'; TextOff 'Messages / Meldungen'
      on Click: ActivateScreen("20_Messages", 0)
      Appearance <- "MainNavigationState"
   Button "Button_3" at 0,201 size 220x60; TextOn 'Menu Item 3'; TextOff 'Diagnostics / Diagnose'
      on Click: ActivateScreen("30_Diagnostics", 0)
      Appearance <- "MainNavigationState"
   Rectangle "Rectangle_1" at 214,78 size 6x60
      Visibility <- "MainNavigationState"
   Rectangle "Rectangle_2" at 214,140 size 6x60
      Visibility <- "MainNavigationState"
   Rectangle "Rectangle_3" at 214,201 size 6x60
      Visibility <- "MainNavigationState"
   Button "Button_4" at 0,262 size 220x60; TextOn 'Menu Item 4'; TextOff 'Settings / Einstellungen'
      on Click: ActivateScreen("40_Settings", 0)
      Appearance <- "MainNavigationState"
   Rectangle "Rectangle_4" at 214,262 size 6x60
      Visibility <- "MainNavigationState"

VB script "ActivateAlarmControlScreen"
   bec8f1e5-2ab1-45f6-ad91-1d37c469eb91 20_Messages,0

VB script "ActivateStartScreen"
   HmiRuntime.BaseScreenName = SmartTags("StartScreenName")

VB script "CheckCurrentLanguage"
   If HmiRuntime.Language = 1031 Then 'German
   	SmartTags("CurrentLanguage") = 0
   	ElseIf HmiRuntime.Language = 1033 Then 'English US
   	SmartTags("CurrentLanguage") = 1
   End If
   
   	

VB script "CheckCurrentUserName"
   If SmartTags("CurrentUserName") = "" Or SmartTags("CurrentUserName") = "User Name" Or SmartTags("CurrentUserName") = "Benutzer" Then
     
     If HmiRuntime.Language = 1031 Then 'Germany
       SmartTags("CurrentUserName") = "Benutzer"
       
     ElseIf HmiRuntime.Language = 1033 Then 'English US
       SmartTags("CurrentUserName") = "User Name"
     End If
     
     SmartTags("UserIsLoggedIn") = False
   Else
     If SmartTags("CurrentUserName") <> "User Name" And SmartTags("CurrentUserName") <> "Benutzer" Then
       SmartTags("UserIsLoggedIn") = True  
     End If
   End If

VB script "CheckDiagState"
   If SmartTags("@DiagnosticsIndicatorTag") = 1 Then
   	SmartTags("DiagState") = 1
   Else
   	SmartTags("DiagState") = 0
   End If

VB script "GetStartScreenName"
   SmartTags("StartScreenName") = HmiRuntime.BaseScreenName

VB script "ShowLoginPopUp"
   efd93a16-2665-4b85-bcb9-25eddcb7b6f4 Template_Logon_Logoff,250,30,$3$hmiOn$,$3$hmiAnimationOff$,$3$hmiFast$

VB script "ShowOperatingModePopUp"
   efd93a16-2665-4b85-bcb9-25eddcb7b6f4 Template_Operating_Mode,188,30,$3$hmiOn$,$3$hmiAnimationOff$,$3$hmiFast$

VB script "ShowOptionPanelPopUp"
   efd93a16-2665-4b85-bcb9-25eddcb7b6f4 OptionPanel_4_Buttons, 410, 104, $3$hmiOn$, $3$hmiRight$, $3$hmiFast$

VB script "ShowRecipePopUp"
   efd93a16-2665-4b85-bcb9-25eddcb7b6f4 Template_Recipe,50,30,$3$hmiOn$,$3$hmiAnimationOff$,$3$hmiFast$

scheduled task "User Name"
   on Action: function_f41c6f6c("CurrentUserName"); "CheckCurrentUserName"()
*)